FUNCTION_BLOCK FB_LamparaComputada_IL
VAR_INPUT
    Reinicia: BOOL;
    ManiobrasTotales: UINT := 2;
    TiempoEncendido: REAL := 2.0;
END_VAR
VAR_OUTPUT
    Habilitada: BOOL;
    ManiobrasPendientes: UINT;
    TiempoPendiente: REAL;
END_VAR
VAR
    Lampara AT %Q*: BOOL;
    Pulsador AT %I*: BOOL;
    
    Temporizador: TON;
    Contador: CTD;
    Memoria: RS;

    Resultado: REAL;
    Tiempo: TIME;
END_VAR

// NETWORK 1
// instruction list
LD      TiempoEncendido
MUL     1000
ST      Resultado

// NETWORK 2
// instruction list
LD      Resultado
REAL_TO_TIME
ST      Tiempo

// NETWORK 3
// instruction list
CAL     Temporizador(
    IN      := Lampara,
    PT      := Tiempo)

// NETWORK 4
// instruction list
CAL     Contador(
    CD      := Lampara,
    LOAD    := Reinicia,
    PV      := ManiobrasTotales)

// NETWORK 5
// instruction list
LDN     Contador.Q
ST      Habilitada

// NETWORK 6
// instruction list
LD      Contador.CV
ST      ManiobrasPendientes

// NETWORK 7
// instruction list
LD      Habilitada
AND     Pulsador
S       Lampara

// NETWORK 8
// instruction list
LD      Temporizador.Q
R       Lampara

// NETWORK 9
// instruction list
LD      Temporizador.ET
TIME_TO_REAL
ST      Resultado

// NETWORK 10
// instruction list
LD      Resultado
DIV     1000
ST      Resultado

// NETWORK 11
// instruction list
LD      TiempoEncendido
SUB     Resultado
ST      TiempoPendiente

// NETWORK 12
// instruction list

END_FUNCTION_BLOCK

(* stored: Version 1.1.0.1, ProductVersion 3.1.4024.12
   POU FB_LamparaComputada_IL: Id {6a650317-49f9-46df-a598-4c9e5c8c1170}, SpecialFunc None *)
